{attribute 'GeneratedUsingTerminal: EL6201-0000-0017'}
{attribute addProperty BoxType "EL6201-0000-0017"}
{attribute addProperty Id "Slave_1A_DO0BOOL1Slave_1A_DO1BOOL1Slave_1A_DO2BOOL1Slave_1A_DO3BOOL1Slave_1B_DO0BOOL1Slave_1B_DO1BOOL1Slave_1B_DO2BOOL1Slave_1B_DO3BOOL1"}
{attribute addProperty CRC "2181705981"}
{attribute addProperty Size "8"}
TYPE Slave_1_Outputs_820A30FD :
STRUCT
	{attribute addProperty Name "Slave_1A_DO0"}
	Slave_1A_DO0 : BOOL;
	{attribute addProperty Name "Slave_1A_DO1"}
	Slave_1A_DO1 : BOOL;
	{attribute addProperty Name "Slave_1A_DO2"}
	Slave_1A_DO2 : BOOL;
	{attribute addProperty Name "Slave_1A_DO3"}
	Slave_1A_DO3 : BOOL;
	{attribute addProperty Name "Slave_1B_DO0"}
	Slave_1B_DO0 : BOOL;
	{attribute addProperty Name "Slave_1B_DO1"}
	Slave_1B_DO1 : BOOL;
	{attribute addProperty Name "Slave_1B_DO2"}
	Slave_1B_DO2 : BOOL;
	{attribute addProperty Name "Slave_1B_DO3"}
	Slave_1B_DO3 : BOOL;
END_STRUCT
END_TYPE

(* stored: Version 1.2.0.0, ProductVersion 3.1.4024.9
   DUT Slave_1_Outputs_820A30FD: Id {aba90e5c-28b3-4772-8d14-cac7ae330c22} *)
